// Object representing a conveyor lane consisting of multiple zones
FUNCTION_BLOCK FB_SeqConveyorLane
(************************************************************************************** 
* 	Application 		: BoxControl Framework 
* 	Revision 			: $Revision: 404877 $ 
* 	Revision date 		: $Date: 2018-04-26 14:10:34 +0200 (Thu, 26 Apr 2018) $ 
* 	Last changed by 	: $Author: b7ernsb $ 
* 	URL 				: $URL: http://almscdc.swisslog.com/repo/SWPD/Development/BoxControlFramework/21_Projects/BCF_2.0/trunk/BCF/BCF/JumpStart/20_Product/10_App/12_E_Functions/10_Lib/10_Conv/FB_FunctionConv.TcPOU $ 
* ------------------------------------------------------------------------------------ 
* 	© Swisslog AG 
* 	Swisslog is not liable for any usage of this source code that is not agreed 
* 	on between Swisslog and the other party. The mandatory legal liability remains 
* 	unaffected. 
* ------------------------------------------------------------------------------------ 
* 	Revision History: 
* 
* 	VERSION 		DATE 			INITIALS 			DESCRIPTION 
* 	0.1 			06.05.2019 		ber 				Created.

* 
**************************************************************************************)
VAR_INPUT
	Positions						: ARRAY [1..MAX_LANE_SIZE] OF ST_PositionIdent; // Index 1: Outfeed position of the lane 
END_VAR
VAR
	PositionCount					: DINT; // Amount of positions in the lane
	OnlySequencingTU				: BOOL:= TRUE; // Only allow TU with sequencing data to enter the lane
	Idx								: DINT;
END_VAR

VAR CONSTANT
	MAX_LANE_SIZE					: DINT:=SequencingParameter.MAX_LANE_SIZE; // Maximal number of zones in a conveyor lane
END_VAR

PositionCount:= 0;	
// Determine amount of positions in the lane
FOR Idx:=1 TO MAX_LANE_SIZE DO
	IF Positions[Idx].eFunctionNumber>0 THEN
		PositionCount:= PositionCount+1;
	END_IF
END_FOR

/// Returns all TU indices currently present in the lane
METHOD M_GetAllTU : BOOL // True = execution sucessfull, else false
VAR_IN_OUT
	mTU_Indices	: ARRAY [*] OF DINT; // List of all TU data indices in the lane
END_VAR
VAR
	mIdx		: DINT;
	mTU_Index	: DINT;
	mCount		: DINT;
END_VAR
MEMSET(ADR(mTU_Indices^), 0,  DINT_TO_UDINT((UPPER_BOUND(mTU_Indices,1)- LOWER_BOUND(mTU_Indices,1)+1)*SIZEOF(mTU_Indices^)));	
mCount:= LOWER_BOUND(mTU_Indices,1);
M_GetAllTU:= TRUE;	

// Loop through lane
FOR mIdx:=1 TO PositionCount DO	
	
	mTU_Index:= F_GetTU_DataIndex(Positions[mIdx].eFunctionNumber, Positions[mIdx].ZoneNumber);
	
	// If a TU index is present on the zone	
	IF mTU_Index > 0 THEN

		// Input array has enough space
		IF mCount <= UPPER_BOUND( mTU_Indices,1) THEN
			
			mTU_Indices[mCount]:= mTU_Index;
			mCount:= mCount+1;
		
		ELSE // Input array too small
	
			MEMSET(ADR(mTU_Indices^), 0, DINT_TO_UDINT((UPPER_BOUND(mTU_Indices,1)- LOWER_BOUND(mTU_Indices,1)+1)*SIZEOF(mTU_Indices^)));		
			M_GetAllTU:= FALSE;	
			EXIT;		
		END_IF

	END_IF
END_FOR
END_METHOD

// Get TU Index on first occupied position (nearest to the infeed)
METHOD M_GetFirstTU : DINT // TU index
VAR
	mIdx				: DINT;
END_VAR
VAR_INST
	TransportCtrlData	: ST_TransportControlData;	
END_VAR
M_GetFirstTU:=0;

// Loop through lane from infeed to outfeed
FOR mIdx:=0 TO PositionCount-1 DO	
	
	TransportCtrlData:= F_GetTransportControlData(Positions[PositionCount-mIdx].eFunctionNumber, Positions[PositionCount-mIdx].ZoneNumber);

	// Finish search when a TU was found	
	IF  TransportCtrlData.NumberOfPresentTUs > 0 THEN
		M_GetFirstTU:=F_GetTU_DataIndex( Positions[PositionCount-mIdx].eFunctionNumber, Positions[PositionCount-mIdx].ZoneNumber);
		EXIT;
	END_IF
	
END_FOR
END_METHOD

// Get TU Index on last occupied position (nearest to the outfeed)
METHOD M_GetLastTU : DINT // TU index
VAR
	mIdx				: DINT;
END_VAR
VAR_INST
	TransportCtrlData	: ST_TransportControlData;	
END_VAR
M_GetLastTU:=0;

// Loop through lane from outfeed to infeed
FOR mIdx:=1 TO PositionCount DO	
	
	TransportCtrlData:= F_GetTransportControlData(Positions[mIdx].eFunctionNumber, Positions[mIdx].ZoneNumber);
	
	// Finish search when a TU was found
	IF  TransportCtrlData.NumberOfPresentTUs > 0 THEN
		M_GetLastTU:= F_GetTU_DataIndex( Positions[mIdx].eFunctionNumber, Positions[mIdx].ZoneNumber);
		EXIT;
	END_IF
	
END_FOR
END_METHOD

// Returns number of empty zones in the lane
METHOD M_GetNrOfEmptyZones : DINT 
VAR
	mIdx				: DINT;
	mEmptyPosition_Count: DINT;
END_VAR
VAR_INST
	TransportCtrlData	: ST_TransportControlData;	
END_VAR
// Loop through lane from outfeed to infeed
FOR mIdx:=1 TO PositionCount DO	
	
	TransportCtrlData:= F_GetTransportControlData(Positions[mIdx].eFunctionNumber, Positions[mIdx].ZoneNumber);
	
	// Increase count when no TU is present on the zone
	IF  TransportCtrlData.NumberOfPresentTUs = 0 THEN
		mEmptyPosition_Count:=mEmptyPosition_Count+1;
	END_IF
	
END_FOR

M_GetNrOfEmptyZones:= mEmptyPosition_Count;
END_METHOD

// Returns number of occupied zones in the lane
METHOD M_GetNrOfOccupiedZones : DINT 
VAR
	mIdx				: DINT;
	mTU_Count			: DINT;
END_VAR
VAR_INST
	TransportCtrlData	: ST_TransportControlData;	
END_VAR
// Loop through lane from outfeed to infeed
FOR mIdx:=1 TO PositionCount DO	
	
	TransportCtrlData:= F_GetTransportControlData(Positions[mIdx].eFunctionNumber, Positions[mIdx].ZoneNumber);

	// Increase count when TU is present on the zone	
	IF  TransportCtrlData.NumberOfPresentTUs > 0 THEN
		mTU_Count:=mTU_Count+1;
	END_IF
	
END_FOR

M_GetNrOfOccupiedZones:= mTU_Count;
END_METHOD

/// Returns all TU indices (which have sequencing data)  after the last sequence error (sequence error nearest to the lane outfeed)
METHOD M_GetTUs_AfterLastError : BOOL; // True = execution successfull, else false
VAR_IN_OUT
	mTU_Indices					: ARRAY [*] OF DINT; // List of TU data indices after the error
	mTU_Table					: ARRAY[0..Conveyor.NUMBER_OF_TU_DATA] OF ST_TU_Data; // TU Table
END_VAR
VAR 
	mIdx						: DINT;
	mTU_IdxTemp					: DINT;
	mTU_IdxOutput				: DINT; 
	mCount						: DINT;
	mSequenceErrorFound			: BOOL;
END_VAR
VAR_INST
	TransportCtrlDataOutput		: ST_TransportControlData; 
	TransportCtrlDataTemp		: ST_TransportControlData; 
END_VAR
MEMSET(ADR(mTU_Indices^), 0, DINT_TO_UDINT((UPPER_BOUND(mTU_Indices,1)- LOWER_BOUND(mTU_Indices,1)+1)*SIZEOF(mTU_Indices^)));		
M_GetTUs_AfterLastError:=TRUE;
mCount:= LOWER_BOUND(mTU_Indices,1);

// Loop through lane
FOR mIdx:=1 TO PositionCount DO
	
	TransportCtrlDataTemp:= F_GetTransportControlData(Positions[mIdx].eFunctionNumber, Positions[mIdx].ZoneNumber);
	mTU_IdxTemp:= F_GetTU_DataIndex(Positions[mIdx].eFunctionNumber, Positions[mIdx].ZoneNumber);

	// Check if there is TU with sequencing information	
	IF  TransportCtrlDataTemp.NumberOfPresentTUs > 0 AND mTU_Table[mTU_IdxTemp].DataSet.Sequence > 0 THEN
		
		// New TU  with sequencing data found		
		IF mTU_IdxOutput = 0 THEN
			
			// Set TU as comparable
			mTU_IdxOutput := mTU_IdxTemp;
			TransportCtrlDataOutput:= TransportCtrlDataTemp;
		
		// Check if both TUs have the same destination ( belong to the same stream).	
		ELSIF  mTU_Table[mTU_IdxOutput].Destination[1].eFunctionNumber <> mTU_Table[mTU_IdxTemp].Destination[1].eFunctionNumber OR
				mTU_Table[mTU_IdxOutput].Destination[1].ZoneNumber <> mTU_Table[mTU_IdxTemp].Destination[1].ZoneNumber OR
				mTU_Table[mTU_IdxOutput].DataSet.DestinationSlot <> mTU_Table[mTU_IdxTemp].DataSet.DestinationSlot THEN
		
			// TUs dont belong to the same stream!!
			M_GetTUs_AfterLastError:=FALSE;
			EXIT;	
				
		
		ELSE // Compare with TU nearer to the output		
		
			// Check if TU which is nearer to the output is located higher in the stream	
			IF	mTU_Table[mTU_IdxOutput].DataSet.Sequence >  mTU_Table[mTU_IdxTemp].DataSet.Sequence OR 
				(mTU_Table[mTU_IdxOutput].DataSet.Sequence =  mTU_Table[mTU_IdxTemp].DataSet.Sequence AND
				mTU_Table[mTU_IdxOutput].DataSet.SubSequence >  mTU_Table[mTU_IdxTemp].DataSet.SubSequence)THEN				
				
				// Sequence error detected
				mSequenceErrorFound:= TRUE;
				EXIT;
				
			ELSE // TUs are in correct sequencing order
	
				// Set TU as new comparable
				mTU_IdxOutput := mTU_IdxTemp;
				TransportCtrlDataOutput:= TransportCtrlDataTemp;			
			END_IF	
		END_IF
		
		// If input list is big enough, add the found index
		IF  mCount <= UPPER_BOUND(mTU_Indices,1) THEN
				
			// Add index to list
			mTU_Indices[mCount]:= mTU_IdxTemp;
			mCount:= mCount+1;
				
		ELSE // Array too small
			M_GetTUs_AfterLastError:=FALSE;
			EXIT;
		END_IF
		
	END_IF
END_FOR


IF NOT mSequenceErrorFound OR NOT M_GetTUs_AfterLastError THEN
	MEMSET(ADR(mTU_Indices^), 0, DINT_TO_UDINT((UPPER_BOUND(mTU_Indices,1)- LOWER_BOUND(mTU_Indices,1)+1)*SIZEOF(mTU_Indices^)));		
END_IF
END_METHOD

/// Checks if there is a sequence error pending  within the lane
METHOD M_HasSquenceError : BOOL // True = sequence error pending, else false
VAR_IN_OUT
	mTU_Table					: ARRAY[0..Conveyor.NUMBER_OF_TU_DATA] OF ST_TU_Data; // TU Data Table
END_VAR
VAR 
	mTU_IdxTemp					: DINT;
	mTU_IdxOutput				: DINT; 
	mIdx						: DINT;
	mSequenceErrorFound			: BOOL;
END_VAR
VAR_INST
	TransportCtrlDataOutput		: ST_TransportControlData; 
	TransportCtrlDataTemp		: ST_TransportControlData;
END_VAR
mSequenceErrorFound:=FALSE;

// Loop through lane from outfeed to infeed
FOR mIdx:=1 TO PositionCount DO
	
	TransportCtrlDataTemp:= F_GetTransportControlData(Positions[mIdx].eFunctionNumber, Positions[mIdx].ZoneNumber);
	mTU_IdxTemp:= F_GetTU_DataIndex(Positions[mIdx].eFunctionNumber, Positions[mIdx].ZoneNumber);

	// Check if there is TU with sequencing information	
	IF  TransportCtrlDataTemp.NumberOfPresentTUs > 0 AND mTU_Table[mTU_IdxTemp].DataSet.Sequence > 0 THEN
		
		// New TU  with sequencing data found		
		IF mTU_IdxOutput = 0 THEN
			
			// Set TU as comparable
			mTU_IdxOutput := mTU_IdxTemp;
			TransportCtrlDataOutput:= TransportCtrlDataTemp;
		
		// Check if both TUs have the same destination ( belong to the same stream).	
		ELSIF  mTU_Table[mTU_IdxOutput].Destination[1].eFunctionNumber <> mTU_Table[mTU_IdxTemp].Destination[1].eFunctionNumber OR
				mTU_Table[mTU_IdxOutput].Destination[1].ZoneNumber <> mTU_Table[mTU_IdxTemp].Destination[1].ZoneNumber OR
				mTU_Table[mTU_IdxOutput].DataSet.DestinationSlot <> mTU_Table[mTU_IdxTemp].DataSet.DestinationSlot THEN
		

			mSequenceErrorFound:=TRUE;
			EXIT;	
				
		
		ELSE // Compare with TU nearer to the output		
		
			// Check if TU which is nearer to the output is located higher in the stream	
			IF	mTU_Table[mTU_IdxOutput].DataSet.Sequence >  mTU_Table[mTU_IdxTemp].DataSet.Sequence OR 
				(mTU_Table[mTU_IdxOutput].DataSet.Sequence =  mTU_Table[mTU_IdxTemp].DataSet.Sequence AND
				mTU_Table[mTU_IdxOutput].DataSet.SubSequence >  mTU_Table[mTU_IdxTemp].DataSet.SubSequence)THEN				
				

				mSequenceErrorFound:= TRUE;
				EXIT;
				
			ELSE // TUs are in correct sequencing order
	
				// Set TU as new comparable
				mTU_IdxOutput := mTU_IdxTemp;
				TransportCtrlDataOutput:= TransportCtrlDataTemp;
			END_IF		
		END_IF
	END_IF
END_FOR


M_HasSquenceError:= mSequenceErrorFound;
END_METHOD

METHOD M_IsEmpty : BOOL // True = lane is empty, otherwise false
VAR
	mIdx				: DINT;
	mTransportCtrlData	: ST_TransportControlData;
END_VAR
M_IsEmpty:= TRUE;

// Loop through lane from outfeed to infeed
FOR mIdx:=1 TO PositionCount DO	
	
	mTransportCtrlData:= F_GetTransportControlData(Positions[mIdx].eFunctionNumber, Positions[mIdx].ZoneNumber);

	// Finish search when a TU was found		
	IF mTransportCtrlData.NumberOfPresentTUs > 0 THEN
		M_IsEmpty:= FALSE;
		EXIT;
	END_IF
	
END_FOR
END_METHOD

METHOD M_IsFull : BOOL // True = lane is full, otherwise false
VAR
	mIdx				: DINT;
	mTransportCtrlData	: ST_TransportControlData;
END_VAR
M_IsFull:= TRUE;

// Loop through lane from outfeed to infeed
FOR mIdx:=1 TO PositionCount DO	
	
	mTransportCtrlData:= F_GetTransportControlData(Positions[mIdx].eFunctionNumber, Positions[mIdx].ZoneNumber);

	// Finish search when a TU an empty zone was found	
	IF mTransportCtrlData.NumberOfPresentTUs = 0 THEN
		M_IsFull:= FALSE;
		EXIT;
	END_IF
	
END_FOR
END_METHOD

/// Check if TU may enter the lane, depening on  sequence information
METHOD M_RequestAccess : BOOL // True = Access granted, else false
VAR_INPUT
	mTU_Index			: DINT; // TU data index of requesting TU
END_VAR
VAR_IN_OUT 
	mTU_Table			: ARRAY[0..Conveyor.NUMBER_OF_TU_DATA] OF ST_TU_Data; // TU Table
END_VAR
VAR
	mIdx				: DINT;
	mTU_IndexLane		: DINT;
END_VAR
VAR_INST
	TransportCtrlData	: ST_TransportControlData;	
END_VAR
M_RequestAccess:=FALSE;	

IF M_IsEmpty() THEN

	// Grant access if TU has sequencing data or non sequencing TU's are allowed by configuration
	IF  mTU_Table[mTU_Index].DataSet.Sequence > 0 OR  NOT OnlySequencingTU THEN
		M_RequestAccess:=TRUE;	
	END_IF
	
ELSIF M_IsFull() THEN
	; //  Deny access

// Lane is partially full and requesting TU has no  sequencing data	
ELSIF  mTU_Table[mTU_Index].DataSet.Sequence = 0  THEN
		
	IF  NOT OnlySequencingTU THEN
		M_RequestAccess:= TRUE;
	END_IF

ELSE // Lane is partially full and requesting TU has data	
	
	// Search first TU after lane input with sequencing information
	FOR mIdx:=0 TO PositionCount-1 DO	

		TransportCtrlData:= F_GetTransportControlData(Positions[PositionCount-mIdx].eFunctionNumber, Positions[PositionCount-mIdx].ZoneNumber);
		mTU_IndexLane:= F_GetTU_DataIndex(Positions[PositionCount-mIdx].eFunctionNumber, Positions[PositionCount-mIdx].ZoneNumber);
	
		// Only consider TUs with whose Sequencing is not on hold
		IF TransportCtrlData.NumberOfPresentTUs > 0 AND 
			NOT mTU_Table[mTU_IndexLane].DataSet.HaltSequencing THEN
			
			 // Check if requesting TU is located higher in the stream (lower priority) than the found TU  
			IF  mTU_Table[mTU_Index].Destination[1].eFunctionNumber = mTU_Table[mTU_IndexLane].Destination[1].eFunctionNumber AND
				mTU_Table[mTU_Index].Destination[1].ZoneNumber = mTU_Table[mTU_IndexLane].Destination[1].ZoneNumber AND
				mTU_Table[mTU_Index].DataSet.DestinationSlot = mTU_Table[mTU_IndexLane].DataSet.DestinationSlot AND
				mTU_Table[mTU_Index].DataSet.Sequence >  mTU_Table[mTU_IndexLane].DataSet.Sequence OR 
				(mTU_Table[mTU_Index].DataSet.Sequence =  mTU_Table[mTU_IndexLane].DataSet.Sequence AND
				mTU_Table[mTU_Index].DataSet.SubSequence >  mTU_Table[mTU_IndexLane].DataSet.SubSequence)THEN	
								
				M_RequestAccess:= TRUE;				
			END_IF
			
			EXIT;	
			
		END_IF	
	END_FOR
END_IF
END_METHOD

// Only allow TU's to enter the lane which have sequencing data 
PROPERTY P_OnlySequencingTU : BOOL
GET
P_OnlySequencingTU:= OnlySequencingTU;
END_GET
SET
OnlySequencingTU:= P_OnlySequencingTU;
END_SET
END_PROPERTY

END_FUNCTION_BLOCK

(* stored: Version 1.1.0.1, ProductVersion 3.1.4022.12
   POU FB_SeqConveyorLane: Id {f2a4e1b5-9c21-4a06-939c-75a8ae4a4ba3}, SpecialFunc None
   Method M_GetAllTU: Id {4edfffa6-51a2-46d8-ac84-b8079484733f}
   Method M_GetFirstTU: Id {c505bf31-6f37-438e-99f3-1e8a9cbfefff}
   Method M_GetLastTU: Id {cf7f95eb-3f52-4f7d-a335-f5ba9d2d567d}
   Method M_GetNrOfEmptyZones: Id {cd2dbe80-4d77-402b-92ba-cdb13411e46b}
   Method M_GetNrOfOccupiedZones: Id {d2b1253d-5519-46e7-8e98-82d18b0ec7cc}
   Method M_GetTUs_AfterLastError: Id {7e3b6f05-9b01-4036-a468-b61311b0f663}
   Method M_HasSquenceError: Id {aec6bc12-a8cd-4336-b869-3430446eb108}
   Method M_IsEmpty: Id {20b880e5-2790-4846-8580-8e6dcad7066e}
   Method M_IsFull: Id {156c869b-1ea7-4296-a80c-3ab2c73798d9}
   Method M_RequestAccess: Id {f082e898-bd08-4423-a208-bc73d77b425e}
   Property P_OnlySequencingTU: Id {1a6dab28-d059-4c20-aff3-48c19d2ad02d}
   Get Get: Id {536eb5b1-8209-4925-b591-a34e9247ec93}
   Set Set: Id {505afa7a-9461-47fc-848c-6727535d85e2} *)
